INTERFACE I_DatatypeAddedEvent EXTENDS I_Event

PROPERTY PUBLIC Target : I_Datatype
GET
END_GET
END_PROPERTY

END_INTERFACE

(* stored: Version 1.1.0.1, ProductVersion 3.1.4024.12
   Itf I_DatatypeAddedEvent: Id {66f5df5b-09a2-0322-120b-34fede72f678}
   Property Target: Id {6e43ea68-16ca-0ac1-1b24-3c7e2fcf4ad1}
   Get Get: Id {70b4b443-31ac-0ad9-1e5f-52dc042bcb8d} *)
